Staubli VAL3: IsFileOK.pgx

public program IsFileOK(bool& x_bRes (dimensions=1))
begin


  x_bRes=false

  //删除急停文件
  call DeleteAlarmFile()


  //读取动作文件是否正确
  call ReadAction(x_bRes)
  if !x_bRes
    popUpMsg("action.txt动作文件不正确")
    logMsg("action.txt动作文件不正确")
    return
  endIf

  //读取配置文件是否正确
  call ReadCfg(x_bRes)
  if !x_bRes
    popUpMsg("configure.txt配置文件不正确")
    logMsg("configure.txt配置文件不正确")
    return
  endIf


  //读取工艺文件是否正确
  call ReadPreset(x_bRes)
  if !x_bRes
    popUpMsg("preset.txt工艺文件不正确")
    logMsg("preset.txt工艺文件不正确")
    return
  endIf


end
